FUNCTION_BLOCK FB_TrafficLightConsumer
VAR
    light : B3TrafficLight_Plc.FB_TrafficLight;
    lastState : INT;
END_VAR

lastState := light.Step();

END_FUNCTION_BLOCK

(* stored: Version 1.1.0.1
   POU FB_TrafficLightConsumer: Id {b0252502-9298-47c3-b334-f340c0df2e0f}, SpecialFunc None *)
